(* IEC 61131-3 sources: AXOpen/src/core/ctrl/src/IxContext, 2 files *)

(* ---- IxContext.st ---- *)
USING ix.framework.rtc;
USING ix.framework.messaging;

NAMESPACE ix.framework.core
    ///<summary>
    /// Provides base for contextualized entry of `ix.framework` application.
    /// This class is abstract and must be inherited.
    ///</summary>
    CLASS PUBLIC ABSTRACT IxContext IMPLEMENTS IIxContext
        VAR PRIVATE
            _openCounter : ULINT;
            _closeCounter : ULINT;
            _identityCounter : ULINT;
            _messagingLevel : eIxMessageCategory;
            _environment : IIxContextEnvironment;
         END_VAR

        ///<summary>
        /// The entry point for the context. The call tree of the context start here and all the logic of given context
        /// must be placed here.
        /// This method must be overridden in derived class.
        ///</summary>
        METHOD PROTECTED ABSTRACT Main END_METHOD

        METHOD PRIVATE Open : ULINT
            _openCounter := _openCounter + ULINT#1;
        END_METHOD

        METHOD PRIVATE Close : ULINT
            _closeCounter := _closeCounter + ULINT#1;
        END_METHOD

        ///<summary>
        /// Runs the cycle of this context. This method must be called cyclically in a PLC task.
        ///</summary>
        METHOD PUBLIC Run
            THIS.Open();
            THIS.Main();
            THIS.Close();
        END_METHOD

        ///<summary>
        /// Gets the value of current context cycle counter.
        ///</summary>
        METHOD PUBLIC OpenCycleCount : ULINT
            OpenCycleCount := _openCounter;
        END_METHOD

        METHOD PUBLIC ClosedCycleCount : ULINT
            ClosedCycleCount := _closeCounter;
        END_METHOD

        METHOD PUBLIC CreateIdentity : ULINT
            _identityCounter := _identityCounter + ULINT#1;
            CreateIdentity := _identityCounter;
        END_METHOD

        METHOD PUBLIC PeekIdentity : ULINT
            PeekIdentity := _identityCounter;
        END_METHOD

        VAR PRIVATE
            NULL_RTC : _NULL_RTC;
            _rtc : IRtc;
        END_VAR

        METHOD PUBLIC GetRtc : IRtc
            IF(_rtc <> NULL) THEN
                GetRtc := _rtc;
            ELSE
                GetRtc := NULL_RTC;
            END_IF;
        END_METHOD

        METHOD PUBLIC InjectRtc
            VAR_INPUT
                Rtc : IRtc;
            END_VAR
            _rtc := Rtc;
        END_METHOD

        METHOD PUBLIC Environment : IIxContextEnvironment
            Environment := _environment;
        END_METHOD

        // METHOD PUBLIC SetContextEnvironment
        //     VAR_INPUT
        //         inContextEnvironnment : IIxContextEnvironment;
        //     END_VAR
        //     _contextEnvironment := inContextEnvironnment;
        // END_METHOD
    END_CLASS

    ///<summary>
    /// Provides an empty RTC object for uninitialized RTC.
    ///</summary>
    CLASS PUBLIC _NULL_RTC IMPLEMENTS IRtc
        VAR PRIVATE
            _null_time : LDATE_AND_TIME := LDATE_AND_TIME#1970-01-01-00:00:00.000;
        END_VAR
        METHOD PUBLIC NowUTC : LDATE_AND_TIME
            NowUTC := _null_time;
        END_METHOD
    END_CLASS
END_NAMESPACE

(* ---- IxContextEnvironment.st ---- *)
USING ix.framework.messaging;

NAMESPACE ix.framework.core
    CLASS PUBLIC IxContextEnvironment IMPLEMENTS IIxContextEnvironment
        VAR PRIVATE
            _messenger : IxMessengerEnv;
        END_VAR
        METHOD PUBLIC Messaging : IIxMessengerEnv
            Messaging := _messenger;
        END_METHOD
    END_CLASS
END_NAMESPACE
